(* IEC 61131-3 sources: ArfBotOS/Codesys-4/ArfBotOS.fbsdev/Application.iecapp^/FUN/FB_ProgramProcessor.fb.st^/private, 1 file *)

(* ---- _M_Error.meth.st ---- *)
METHOD PRIVATE _M_Error
VAR_INPUT
    Description: STRING;
END_VAR

SUPER^.M_Error(Description := CONCAT('Program Processor: ', Description));
END_METHOD
